TYPE ST_EAP_Pub_Variable :
STRUCT
	Name				: 	STRING;		// Name of the Variable
	VarState	AT %I*	:	UINT;		// VarState.0 = Not Sent, 1 = Transmission Suspended, 0 = Transmission OK
	VarID 		AT %Q*	:	UINT;		// Changeable ID of the variable
	VarCtrl		AT %Q*	:	UINT;		// VarCtrl.0 = Disable publishing
END_STRUCT
END_TYPE

(* stored: Version 1.1.0.1, ProductVersion 3.1.4024.6
   DUT ST_EAP_Pub_Variable: Id {a8625ea2-c604-458b-8a6a-622da2114391} *)
